Yaskawa INFORM job: R1_W68-69(-90,-90)KM-OK.JBI

/JOB
//NAME R1_W68-69(-90,-90)KM-OK
///FOLDERNAME KRIS-SCIANA
//POS
///NPOS 49,49,0,4,0,0
///TOOL 0
///POSTYPE PULSE
///PULSE
C00000=59135,-25377,-6981,14089,62612,17507
C00001=62613,-31099,-7610,14128,60942,21463
C00002=59940,-5159,40679,18119,45646,17920
C00003=59624,3615,52643,19120,42998,17213
C00004=59501,7492,57968,19613,41807,16882
C00005=59497,11001,63803,20311,40123,16465
C00006=59501,7492,57968,19613,41807,16882
C00007=70954,12769,60387,-5412,43467,30634
C00008=70094,14241,61747,-5188,43338,30283
C00009=70954,12769,60387,-5412,43467,30634
C00010=70347,15555,62894,1608,41972,27570
C00011=70761,18379,66707,1507,41071,27729
C00012=70116,15192,62802,1683,41847,27470
C00013=70565,11395,57405,1505,43209,27686
C00014=71720,2948,45409,1099,46233,28211
C00015=49054,52400,94850,-59,71875,-26451
C00016=49054,26059,47856,-57,87262,-26459
C00017=49054,27038,49871,-57,86525,-26459
C00018=49972,30482,54726,129,85305,-26164
C00019=49972,31976,57659,129,84268,-26165
C00020=49524,30460,55672,37,84713,-26308
C00021=50449,32645,57909,225,84457,-26012
C00022=51067,34180,59498,350,84267,-25815
C00023=50458,32666,57930,227,84455,-26008
C00024=50458,26424,45164,227,89103,-26000
C00025=64210,3164,44535,3054,77287,-21763
C00026=65385,8893,54563,3336,74023,-21486
C00027=65855,11500,58998,3455,72618,-21383
C00028=65850,14757,64478,3487,70923,-21432
C00029=65855,11500,58998,3455,72618,-21383
C00030=67270,-5278,43106,4072,64273,-19764
C00031=67800,-3359,45419,4130,63814,-19609
C00032=67021,-5448,43284,4059,64088,-19852
C00033=67956,29497,79488,3206,78608,-21982
C00034=68497,31304,83152,3396,77266,-21865
C00035=67484,34034,86095,3072,76890,-22157
C00036=67045,30525,80104,2911,78785,-22235
C00037=65957,23710,67836,2535,82860,-22462
C00038=66976,11986,60686,52108,68160,-17724
C00039=82575,28324,48009,11244,75457,6524
C00040=82590,41711,73928,11473,66498,5822
C00041=66475,9175,56958,51734,68940,-17497
C00042=66263,10146,59005,51903,68560,-17828
C00043=82600,41716,73892,11470,66523,5828
C00044=83787,40706,72849,11512,66488,6228
C00045=92496,27666,59042,-4487,61341,11856
C00046=97139,11107,37515,-4628,66311,13293
C00047=66831,-18265,3169,22895,44504,326
C00048=17826,-159560,-130732,23103,44734,299
BC00000=235821,1066677,863150
BC00001=240034,1062633,854656
BC00002=240034,1062633,854656
BC00003=240034,1062633,854656
BC00004=240034,1062633,854656
BC00005=240034,1062633,854656
BC00006=240034,1062633,854656
BC00007=240034,1062633,854656
BC00008=240034,1062633,854656
BC00009=240034,1062633,854656
BC00010=240034,1062633,854656
BC00011=240034,1062633,854656
BC00012=240034,1062633,854656
BC00013=240034,1062633,854656
BC00014=240034,1062633,854656
BC00015=183955,1027061,855724
BC00016=183955,1027061,731173
BC00017=183955,1027061,731173
BC00018=183955,1027061,731173
BC00019=183955,1027061,731173
BC00020=183955,1027061,731173
BC00021=183955,1027061,731173
BC00022=183955,1027061,731173
BC00023=183955,1027061,731173
BC00024=183955,1027061,731173
BC00025=183955,1027060,855728
BC00026=183955,1027060,855728
BC00027=183955,1027060,855728
BC00028=183955,1027060,855728
BC00029=183955,1027060,855728
BC00030=183955,1027060,855728
BC00031=183955,1027060,855728
BC00032=183955,1027060,855728
BC00033=183955,1027060,855728
BC00034=183955,1027060,855728
BC00035=183955,1027060,855728
BC00036=183955,1027060,855728
BC00037=183955,1027060,855728
BC00038=219769,1097364,867779
BC00039=176237,1102292,771900
BC00040=175875,1102387,772140
BC00041=215924,1089340,738813
BC00042=215924,1089340,738813
BC00043=237622,1102387,772140
BC00044=285781,1102151,772572
BC00045=285781,1102151,772572
BC00046=270113,1102151,772572
BC00047=216950,1076174,898383
BC00048=238915,700065,898383
///POSTYPE BASE
///RECTAN
///RCONF 0,0,0,0,0,0,0,0,0,0,0,0,0,0,0,0,0,0,0,0,0,0,0,0
P00006=0.222,-3.123,-1.508,0.0000,0.0000,0.0000
P00021=-0.225,-6.128,-0.405,0.0000,0.0000,0.0000
P00022=0.222,-3.123,-1.508,0.0000,0.0000,0.0000
P00030=5.926,-4.294,-1.390,0.0000,0.0000,0.0000
//INST
///DATE 2024/07/23 16:05
///ATTR SC,RW
///GROUP1 RB1,BS1
NOP
'r1_W68-69(-90,-90)
'Path S836 (for W508)
SFTOF
MOVJ C00000 BC00000 VJ=100.00
MOVJ C00001 BC00001 VJ=100.00
MOVJ C00002 BC00002 VJ=100.00
MOVJ C00003 BC00003 VJ=100.00
MOVL C00004 BC00004 V=60.0
REFP 3 C00005 BC00005
CALL JOB:SEARCH-R1
SET P021 P006
SFTON P021
MOVL C00006 BC00006 V=60.0
MOVL C00007 BC00007 V=60.0
REFP 3 C00008 BC00008
CALL JOB:SEARCH-R1
SET P021 P006
SFTON P021
MOVL C00009 BC00009 V=60.0
MOVL C00010 BC00010 V=60.0
REFP 3 C00011 BC00011
CALL JOB:SEARCH-R1
SET P021 P006
SFTON P021
MOVL C00012 BC00012 V=60.0
MOVL C00013 BC00013 V=100.0
MOVL C00014 BC00014 V=166.7
'Path S837 (for W508)
SFTOF
MOVL C00015 BC00015 V=1000.0
MOVL C00016 BC00016 V=1000.0
MOVL C00017 BC00017 V=100.0
MOVL C00018 BC00018 V=60.0
REFP 3 C00019 BC00019
CALL JOB:SEARCH-R1
SET P030 P006
SFTON P030
MOVL C00020 BC00020 V=60.0
MOVL C00021 BC00021 V=60.0
REFP 3 C00022 BC00022
CALL JOB:SEARCH-R1
SET P030 P006
SFTON P030
MOVL C00023 BC00023 V=60.0
MOVL C00024 BC00024 V=400.0
SFTOF
MOVL C00025 BC00025 V=166.7
MOVL C00026 BC00026 V=100.0
MOVL C00027 BC00027 V=60.0
REFP 3 C00028 BC00028
CALL JOB:SEARCH-R1
SET P022 P006
SFTON P022
MOVL C00029 BC00029 V=60.0
MOVL C00030 BC00030 V=60.0
REFP 3 C00031 BC00031
CALL JOB:SEARCH-R1
SET P022 P006
SFTON P022
MOVL C00032 BC00032 V=60.0
MOVL C00033 BC00033 V=60.0
REFP 3 C00034 BC00034
CALL JOB:SEARCH-R1
SET P022 P006
SFTON P022
MOVL C00035 BC00035 V=60.0
MOVL C00036 BC00036 V=100.0
MOVL C00037 BC00037 V=400.0
'Path W508
SFTOF
SFTON P022
MOVJ C00038 BC00038 VJ=100.00
MOVJ C00039 BC00039 VJ=100.00
MOVL C00040 BC00040 V=166.7 PL=0
REFP 1 C00041 BC00041
REFP 2 C00042 BC00042
MACRO1 MJ#(0) ARGF9
ARCON
SFTON P030
MOVL C00043 BC00043 V=10.8
SFTON P021
MOVL C00044 BC00044 V=10.8
MOVL C00045 BC00045 V=10.8
ARCOF
MOVL C00046 BC00046 V=333.3
SFTOF
MOVJ C00047 BC00047 VJ=100.00
MOVJ C00048 BC00048 VJ=100.00
END
